PROGRAM MAIN
VAR
// tst axis 1
 	{attribute 'TcLinkTo' := '.nRawEncoderULINT     := TIIB[Term 6 (EL5042)]^FB Inputs Channel 2^Position'}	
	{attribute 'pytmc' := '
        pv: PLC:TST:MOT:VM:01
        field: DESC Simulated Working Motor
    '}
   
    M1: DUT_MotionStage:=(nEnableMode:=ENUM_StageEnableMode.ALWAYS, bPowerSelf:=TRUE);
    fbMotion1 : FB_MotionStage;

// tst axis 2
	{attribute 'TcLinkTo' := '.nRawEncoderULINT     := TIIB[Term 6 (EL5042)]^FB Inputs Channel 1^Position'}
	{attribute 'pytmc' := '
        pv: PLC:TST:MOT:VM:02
        field: DESC Simulated Working Motor
    '}
    
    M2: DUT_MotionStage:=(nEnableMode:=ENUM_StageEnableMode.ALWAYS, bPowerSelf:=TRUE);
    fbMotion2 : FB_MotionStage;
END_VAR

fbMotion1(stMotionStage:= M1);
fbMotion2(stMotionStage:= M2);
M2.bHardwareEnable := TRUE;
M2.bLimitBackwardEnable := TRUE;
M2.bLimitForwardEnable := TRUE;

END_PROGRAM

(* stored: Version 1.1.0.1, ProductVersion 3.1.4022.18
   POU MAIN: Id {bd3474a7-ace7-4912-9a31-41649952a987}, SpecialFunc None *)
